// Core §6.8 — the ladder face of FB_SequenceBase.
//
// A ladder rung has no statement context: a box runs because power reaches it.
// Every step-facing method therefore takes `Run : BOOL` as its FIRST input, wired
// to the rung, and is a no-op when Run is FALSE (a value-returning call yields its
// fail-closed default). That is the only difference from the ST face; the logic
// itself stays in FB_SequenceBase and is reached through SUPER^.
//
// Chains built on this are integer-based state machines: one rung per state,
// gated by EQ(_step, N), with the boxes chained left to right so power flows
// MOVE -> M_Step -> ... -> M_Advance. The rungs dispatch; they do not evaluate
// transitions, so each rung still ends in M_Advance and the OnJump1..3 mapping
// keeps jumps declarative (§6.10).
FUNCTION_BLOCK ABSTRACT FB_SequenceBaseLd EXTENDS FB_SequenceBase
VAR_INPUT
END_VAR
VAR_OUTPUT
END_VAR
VAR
END_VAR

// §6.8 ST-skeleton progression: at the END of a `CASE _step OF` body, commit the
// step's shared transition result. On ADVANCE (or a declared JUMPn) go to the
// mapped next step and clear the step-scoped latches so the new step re-arms — the
// exact guarantee the SFC exit action gave, in one call. NONE stays put. The caller
// passes its successor map; an unmapped result holds the step (safe, visible).
METHOD M_AdvanceLd
VAR_INPUT
	Run : BOOL;
    OnAdvance : INT;               // next step for E_StepResult.ADVANCE
    // Jump targets default to "not used" so the common case reads
    // `M_Advance(OnAdvance := 100);` instead of repeating `OnJump1..3 := -1`.
    // Defaulted METHOD inputs need TwinCAT >= 3.1.4026, so on the legacy 4024
    // target (FRAKTAL_TC3_4024 defined) they are declared without defaults and
    // every argument is passed explicitly. See Params/PL_FraktalCompat.TcGVL.
    {IF defined (FRAKTAL_TC3_4024)}
    OnJump1   : INT;               // next step for JUMP1 (-1 = not used)
    OnJump2   : INT;               // next step for JUMP2 (-1 = not used)
    OnJump3   : INT;               // next step for JUMP3 (-1 = not used)
    {ELSE}
    OnJump1   : INT := -1;         // next step for JUMP1 (-1 = not used)
    OnJump2   : INT := -1;         // next step for JUMP2 (-1 = not used)
    OnJump3   : INT := -1;         // next step for JUMP3 (-1 = not used)
    {END_IF}
END_VAR
IF Run THEN
	SUPER^.M_Advance(OnAdvance := OnAdvance, OnJump1 := OnJump1, OnJump2 := OnJump2, OnJump3 := OnJump3);
END_IF
END_METHOD

// §6.11 publish a decision request — ladder form: `Run` is the rung's power flow.
// FALSE makes the call a no-op.
METHOD M_AskDecisionLd
VAR_INPUT
    Run : BOOL;
    Req : ST_DecisionRequest;
END_VAR
IF Run THEN
    SUPER^.M_AskDecision(Req := Req);
END_IF
END_METHOD

// §6.9(b) named plain-condition wait — ladder form: `Run` is the rung's power flow.
// FALSE makes the call a no-op and returns FALSE.
METHOD M_AwaitLd : BOOL
VAR_INPUT
    Run : BOOL;
    Idx : INT;
    Label : STRING(120);
    Ok : BOOL;
END_VAR
M_AwaitLd := FALSE;
IF Run THEN
    M_AwaitLd := SUPER^.M_Await(Idx := Idx, Label := Label, Ok := Ok);
END_IF
END_METHOD

// §6.11 withdraw the active request — ladder form: `Run` is the rung's power flow.
// FALSE makes the call a no-op.
METHOD M_ClearDecisionLd
VAR_INPUT
    Run : BOOL;
END_VAR
IF Run THEN
    SUPER^.M_ClearDecision();
END_IF
END_METHOD

// §6.10 shared step-exit action — ladder form: `Run` is the rung's power flow.
// FALSE makes the call a no-op.
METHOD M_ClearTransitionLd
VAR_INPUT
    Run : BOOL;
END_VAR
IF Run THEN
    SUPER^.M_ClearTransition();
END_IF
END_METHOD

// §6.1 one-shot completion (finite chains) — ladder form: `Run` is the rung's power flow.
// FALSE makes the call a no-op.
METHOD M_CompleteLd
VAR_INPUT
    Run : BOOL;
END_VAR
IF Run THEN
    SUPER^.M_Complete();
END_IF
END_METHOD

// §3.9 count a good part directly — ladder form: `Run` is the rung's power flow.
// FALSE makes the call a no-op.
METHOD M_CountGoodLd
VAR_INPUT
    Run : BOOL;
END_VAR
IF Run THEN
    SUPER^.M_CountGood();
END_IF
END_METHOD

// declared process wait; NONE holds the step — ladder form: `Run` is the rung's power flow.
// FALSE makes the call a no-op and returns E_StepResult.NONE.
METHOD M_DelayLd : E_StepResult
VAR_INPUT
    Run : BOOL;
    PT : TIME;
END_VAR
M_DelayLd := E_StepResult.NONE;
IF Run THEN
    M_DelayLd := SUPER^.M_Delay(PT := PT);
END_IF
END_METHOD

// §8.11.1 cycle-complete marker — ladder form: `Run` is the rung's power flow.
// FALSE makes the call a no-op and returns FALSE.
METHOD M_EndOfCycleLd : BOOL
VAR_INPUT
    Run : BOOL;
END_VAR
M_EndOfCycleLd := FALSE;
IF Run THEN
    M_EndOfCycleLd := SUPER^.M_EndOfCycle();
END_IF
END_METHOD

// §6.9 first-out fault from a step — ladder form: `Run` is the rung's power flow.
// FALSE makes the call a no-op.
METHOD M_FaultLd
VAR_INPUT
    Run : BOOL;
    Reason : E_Reason;
    DescriptionKey : STRING(255);
END_VAR
IF Run THEN
    SUPER^.M_Fault(Reason := Reason, DescriptionKey := DescriptionKey);
END_IF
END_METHOD

// §3.4.2 run-style pacing gate — ladder form: `Run` is the rung's power flow.
// FALSE makes the call a no-op and returns FALSE.
METHOD M_GateLd : BOOL
VAR_INPUT
    Run : BOOL;
    Steppable : BOOL;
END_VAR
M_GateLd := FALSE;
IF Run THEN
    M_GateLd := SUPER^.M_Gate(Steppable := Steppable);
END_IF
END_METHOD

// §6.1 issue+await one-shot; FALSE when the rung is not powered — ladder form: `Run` is the rung's power flow.
// FALSE makes the call a no-op and returns FALSE.
METHOD M_TryIssueLd : BOOL
VAR_INPUT
    Run : BOOL;
    Steppable : BOOL;
END_VAR
M_TryIssueLd := FALSE;
IF Run THEN
    M_TryIssueLd := SUPER^.M_TryIssue(Steppable := Steppable);
END_IF
END_METHOD

// §6.12 join of a parallel step — ladder form: `Run` is the rung's power flow.
// FALSE makes the call a no-op and returns NONE.
METHOD M_ParJoinLd : E_StepResult
VAR_INPUT
    Run : BOOL;
END_VAR
M_ParJoinLd := E_StepResult.NONE;
IF Run THEN
    M_ParJoinLd := SUPER^.M_ParJoin();
END_IF
END_METHOD

// §3.16.3 verdict + disposition — ladder form: `Run` is the rung's power flow.
// FALSE makes the call a no-op and returns FALSE.
METHOD M_PartProcessedLd : BOOL
VAR_INPUT
    Run : BOOL;
    Verdict : E_Verdict;
    Reason : E_Reason;
END_VAR
M_PartProcessedLd := FALSE;
IF Run THEN
    M_PartProcessedLd := SUPER^.M_PartProcessed(Verdict := Verdict, Reason := Reason);
END_IF
END_METHOD

// §3.16.3 part received — ladder form: `Run` is the rung's power flow.
// FALSE makes the call a no-op and returns FALSE.
METHOD M_PartReceivedLd : BOOL
VAR_INPUT
    Run : BOOL;
END_VAR
M_PartReceivedLd := FALSE;
IF Run THEN
    M_PartReceivedLd := SUPER^.M_PartReceived();
END_IF
END_METHOD

// §3.16.1 measured value — ladder form: `Run` is the rung's power flow.
// FALSE makes the call a no-op and returns FALSE.
METHOD M_PartRecordLd : BOOL
VAR_INPUT
    Run : BOOL;
    RecordName : STRING(64);
    Value : LREAL;
    Minimum : LREAL;
    Maximum : LREAL;
    Target : LREAL;
    EngUnit : STRING(16);
END_VAR
M_PartRecordLd := FALSE;
IF Run THEN
    M_PartRecordLd := SUPER^.M_PartRecord(RecordName := RecordName, Value := Value, Minimum := Minimum, Maximum := Maximum, Target := Target, EngUnit := EngUnit);
END_IF
END_METHOD

// §3.16.3 processing started — ladder form: `Run` is the rung's power flow.
// FALSE makes the call a no-op.
METHOD M_PartStartedLd
VAR_INPUT
    Run : BOOL;
END_VAR
IF Run THEN
    SUPER^.M_PartStarted();
END_IF
END_METHOD

// §6.9/§8.8 raise a message this step defines itself — ladder form: `Run` is the rung's power flow.
// FALSE makes the call a no-op and returns FALSE.
METHOD M_RaiseCustomLd : BOOL
VAR_INPUT
    Run : BOOL;
    Reason : E_Reason;
    DescriptionKey : STRING(255);
    Severity : E_Severity;
    Category : E_Category;
    LinkPath : STRING(255);
END_VAR
M_RaiseCustomLd := FALSE;
IF Run THEN
    M_RaiseCustomLd := SUPER^.M_RaiseCustom(Reason := Reason, DescriptionKey := DescriptionKey, Severity := Severity, Category := Category, LinkPath := LinkPath);
END_IF
END_METHOD

// §6.9 adopt a child's first-out from conditional step logic — ladder form: `Run` is the rung's power flow.
// FALSE makes the call a no-op and returns FALSE.
METHOD M_RaiseFromChildLd : BOOL
VAR_INPUT
    Run : BOOL;
    Source : I_Module;
END_VAR
M_RaiseFromChildLd := FALSE;
IF Run THEN
    M_RaiseFromChildLd := SUPER^.M_RaiseFromChild(Source := Source);
END_IF
END_METHOD

// §6.9(e) non-blocking custom message — ladder form: `Run` is the rung's power flow.
// FALSE makes the call a no-op and returns FALSE.
METHOD M_RaiseWarningLd : BOOL
VAR_INPUT
    Run : BOOL;
    Reason         : E_Reason;
    DescriptionKey : STRING(255);
    Severity       : E_Severity;
    Category       : E_Category;
END_VAR
M_RaiseWarningLd := FALSE;
IF Run THEN
    M_RaiseWarningLd := SUPER^.M_RaiseWarning(Reason := Reason,
        DescriptionKey := DescriptionKey, Severity := Severity, Category := Category);
END_IF
END_METHOD

// §6.9(e) report a child's failure without adopting it — ladder form: `Run` is
// the rung's power flow. FALSE makes the call a no-op and returns FALSE.
METHOD M_ReportFromChildLd : BOOL
VAR_INPUT
    Run : BOOL;
    Source : I_Module;
END_VAR
M_ReportFromChildLd := FALSE;
IF Run THEN
    M_ReportFromChildLd := SUPER^.M_ReportFromChild(Source := Source);
END_IF
END_METHOD

// §6.12 run one leg of a parallel step — ladder form: `Run` is the rung's power
// flow. FALSE makes the call a no-op and returns FALSE.
METHOD M_RunParLd : BOOL
VAR_INPUT
    Run : BOOL;
    Chain : REFERENCE TO FB_SequenceBase;
    BaseStepNo : INT;
    Branch : INT;
END_VAR
M_RunParLd := FALSE;
IF Run THEN
    M_RunParLd := SUPER^.M_RunPar(Chain := Chain, BaseStepNo := BaseStepNo,
        Branch := Branch);
END_IF
END_METHOD

// §6.8 run another chain as ONE composite step — ladder form: `Run` is the rung's power flow.
// FALSE makes the call a no-op and returns E_StepResult.NONE.
METHOD M_RunSubLd : E_StepResult
VAR_INPUT
    Run : BOOL;
    Chain : REFERENCE TO FB_SequenceBase;
    BaseStepNo : INT;
END_VAR
M_RunSubLd := E_StepResult.NONE;
IF Run THEN
    M_RunSubLd := SUPER^.M_RunSub(Chain := Chain, BaseStepNo := BaseStepNo);
END_IF
END_METHOD

// §6.5 step record + the chart-local ActiveStep mirror, one call.
METHOD M_StepLd
VAR_INPUT
	Run : BOOL;
    StepNo : INT;
    StepName : STRING(120);
    Awaits : I_Module;
    AwaitingLabel : STRING(120);
    TimeClass : E_TimeClass;
    ExpectedTime : TIME;
    // §6.12 concurrent leg; 0 = this chain's own. Required here because a ladder
    // box has no defaulted inputs to omit.
    Branch : INT;
END_VAR
IF Run THEN
	SUPER^.M_Step(StepNo := StepNo, StepName := StepName, Awaits := Awaits, AwaitingLabel := AwaitingLabel, TimeClass := TimeClass, ExpectedTime := ExpectedTime, Branch := Branch);
END_IF
END_METHOD

// §3.4/§8.11 accept the stop between cycles — ladder form: `Run` is the rung's power flow.
// FALSE makes the call a no-op.
METHOD M_StopNowLd
VAR_INPUT
    Run : BOOL;
END_VAR
IF Run THEN
    SUPER^.M_StopNow();
END_IF
END_METHOD

// §3.4 poll at the between-cycles wait — ladder form: `Run` is the rung's power flow.
// FALSE makes the call a no-op and returns FALSE.
METHOD M_StopPendingLd : BOOL
VAR_INPUT
    Run : BOOL;
END_VAR
M_StopPendingLd := FALSE;
IF Run THEN
    M_StopPendingLd := SUPER^.M_StopPending();
END_IF
END_METHOD

// §6.11 consume the answer once (0 = none yet) — ladder form: `Run` is the rung's power flow.
// FALSE makes the call a no-op and returns 0.
METHOD M_TakeDecisionLd : INT
VAR_INPUT
    Run : BOOL;
END_VAR
M_TakeDecisionLd := 0;
IF Run THEN
    M_TakeDecisionLd := SUPER^.M_TakeDecision();
END_IF
END_METHOD

END_FUNCTION_BLOCK

(* stored: Version 1.1.0.1
   POU FB_SequenceBaseLd: Id {51d493b2-6a80-40fc-8489-9750a75237bc}, SpecialFunc None
   Method M_AdvanceLd: Id {347fdf6b-3850-4913-b001-cdea4e2197f1}
   Method M_AskDecisionLd: Id {27b828b7-e6ab-4929-a8e3-bf0128c31e36}
   Method M_AwaitLd: Id {0ab4f7c1-c6cf-445f-8254-00f9b09accae}
   Method M_ClearDecisionLd: Id {ec9bf0d3-47aa-4c63-98ef-c304b344d19c}
   Method M_ClearTransitionLd: Id {e67188a5-fdd7-4322-b6cb-2ada65ea7679}
   Method M_CompleteLd: Id {dd003618-4633-4347-8e9d-013efc953515}
   Method M_CountGoodLd: Id {799295c5-db62-4ed6-bac1-fc03ead3d638}
   Method M_DelayLd: Id {4bf1443b-1271-424b-981d-a7492d5e9705}
   Method M_EndOfCycleLd: Id {30745972-4ddd-43d6-a242-42581b0672aa}
   Method M_FaultLd: Id {4be25263-b392-4c85-9495-75e3d3724ad3}
   Method M_GateLd: Id {3a185ff4-e128-4750-afb7-5cb87585f867}
   Method M_TryIssueLd: Id {d31c61df-3ef5-4878-a4b4-37693736d3c6}
   Method M_ParJoinLd: Id {22213af1-acc1-4d3d-94f0-d19965e3b977}
   Method M_PartProcessedLd: Id {54b056b9-6b46-43fc-9d84-b97f93ca88d3}
   Method M_PartReceivedLd: Id {d4cf9f9b-38f3-4791-b65c-ff9cfdaf4a3f}
   Method M_PartRecordLd: Id {afa5a215-c657-4709-a739-e24817891820}
   Method M_PartStartedLd: Id {50700549-7b3c-41ab-a9af-9dbef655a687}
   Method M_RaiseCustomLd: Id {4a0cdff6-edf4-412a-a7a4-aec736993d6b}
   Method M_RaiseFromChildLd: Id {b5e4c025-e2da-4757-9cd4-7c66992965ee}
   Method M_RaiseWarningLd: Id {25ec3e7d-cdfb-426b-adc5-c48c25344614}
   Method M_ReportFromChildLd: Id {25cd115d-609f-487d-a4a5-11ba53412631}
   Method M_RunParLd: Id {8e30f2f3-d289-4fc3-bdf4-492075436e4a}
   Method M_RunSubLd: Id {ff5366eb-e63d-42b4-9cd8-8aa89d688138}
   Method M_StepLd: Id {eb1b6a4d-878c-4792-a3b6-96b46f1f3886}
   Method M_StopNowLd: Id {d560b992-548f-4361-9200-15082d0c99d1}
   Method M_StopPendingLd: Id {ba7ca419-b2b1-4490-91b8-070539246221}
   Method M_TakeDecisionLd: Id {0ffd832f-1c47-4295-af89-ba583a949b67} *)
